// TIA Portal V18 export
DATA_BLOCK "delaytimes"   // DB52
{ S7_Optimized_Access := 'TRUE' }
VERSION : 0.1
// stored: AutoNumber true, DBAccessibleFromOPCUA true, IsOnlyStoredInLoadMemory false, IsRetainMemResEnabled false, IsWriteProtectedInAS false, MemoryReserve 100
   VAR RETAIN
      "Outlet ON to pump ON A" : Int;
      "Outlet On to pump ON B" : Int;
   END_VAR
   VAR
      "Pump off to Inlet Close A" : Int;
      "Pump off to Inlet Close B" : Int;
   END_VAR
   VAR RETAIN
      "Pump off to Outlet Close" : Int;
      "Mixer ON to outlet ON" : Int;
      "outlet Off to mixer OFF" : Int;
      "Part Present On delay" : DInt;
      "Part Present Off Delay" : DInt;
      "Mixed flowrate error Delay time" : DInt := 2000;
   END_VAR
BEGIN
END_DATA_BLOCK
